Omron CX-Programmer project 新工程 (CX-Programmer 9.73)

# PLC 新PLC1: CPM2* 

## Global symbols (name address type ; comment)
0.00 BOOL  ; 外部急停
0.01 BOOL  ; 自动启动
0.02 BOOL  ; 手动封切
0.03 BOOL  ; 侧推反向磁环
0.04 BOOL  ; 侧推正向磁环
0.05 BOOL  ; 直推反向磁环
0.06 BOOL  ; 直推正向磁环
0.07 BOOL  ; 上膜接近开关
0.08 BOOL  ; 下膜接近开关
0.09 BOOL  ; 封口反向磁环
0.10 BOOL  ; 封口正向磁环
0.11 BOOL  ; 压料反向磁环
10.00 BOOL  ; 侧推电磁阀
10.01 BOOL  ; 直推电磁阀
10.02 BOOL  ; 封口电磁阀
10.03 BOOL  ; 切膜电磁阀
10.04 BOOL  ; 压料电磁阀
10.05 BOOL  ; 上膜电机
10.06 BOOL  ; 下膜电机
10.07 BOOL  ; 送料电机
11.00 BOOL  ; 后送料输出
11.01 BOOL  ; 浮动护栏气缸
11.02 BOOL  ; 一号气缸
11.03 BOOL  ; 二号气缸
11.04 BOOL  ; 三号气缸
11.05 BOOL  ; 四号气缸
11.06 BOOL  ; 熔接输出
11.07 BOOL  ; 熔接瞬间
12.00 BOOL  ; 加热
12.01 BOOL  ; 热风
12.02 BOOL  ; 后输送
12.03 BOOL  ; 报警输出
12.04 BOOL  ; 左右挡板电磁阀
12.05 BOOL  ; 前压料反向电磁阀
13 CHANNEL  ; 套膜包装控制寄存
13.00 BOOL  ; 直推
13.01 BOOL  ; 直推退回
13.02 BOOL  ; 封口
13.03 BOOL  ; 切膜
13.04 BOOL  ; 封膜
13.05 BOOL  ; 气缸复位
13.06 BOOL  ; 后送料启动
14 CHANNEL  ; 自动进料控制寄存
14.00 BOOL  ; 分层/挡料
14.01 BOOL  ; 左右挡板伸出
14.02 BOOL  ; 进料检测
14.03 BOOL  ; 左右挡板回位
14.04 BOOL  ; 顶料上升
14.05 BOOL  ; 末层判断
14.06 BOOL  ; 下一包挡料
14.07 BOOL  ; 左右挡板伸出
14.07 BOOL  ; 顶料下降
14.08 BOOL  ; 侧推
14.09 BOOL  ; 直推
14.10 BOOL  ; 侧推退回
14.11 BOOL  ; 进料完成
16 CHANNEL  ; 气缸输出
17.00 BOOL  ; 一号挡料板
17.01 BOOL  ; 二号挡料板
17.02 BOOL  ; 三号挡料板
17.03 BOOL  ; 四号挡料板
17.04 BOOL  ; 无挡料板
17.08 BOOL  ; 检测第一位
17.09 BOOL  ; 检测第二位
17.10 BOOL  ; 检测第三位
17.11 BOOL  ; 检测第四位
17.12 BOOL  ; 检测第五位
19 CHANNEL  ; 手动封切控制寄存
1.00 BOOL  ; 切膜反向磁环
1.01 BOOL  ; 浮动反向磁环
1.02 BOOL  ; 浮动正向磁环
1.03 BOOL  ; 一号正向磁环
1.04 BOOL  ; 二号正向磁环
1.05 BOOL  ; 三号正向磁环
1.06 BOOL  ; 四号正向磁环
1.07 BOOL  ; 检料光电01
1.08 BOOL  ; 检料光电02
1.09 BOOL  ; 检料接近11
1.10 BOOL  ; 检料接近12
1.11 BOOL  ; 检料光电21
204 CHANNEL  ; 临时整数
20.00 BOOL  ; 文本数据输入
20.01 BOOL  ; 文本数据初始化
20.02 BOOL  ; 文本收缩自动启动
20.03 BOOL  ; 文本收缩自动停止
20.04 BOOL  ; 文本手动封切
20.06 BOOL  ; 文本前送料
20.07 BOOL  ; 文本后送料
20.08 BOOL  ; 文本手动单次进料
20.09 BOOL  ; 文本直推料
20.10 BOOL  ; 文本封口
20.11 BOOL  ; 文本切膜
20.12 BOOL  ; 文本压料
20.13 BOOL  ; 文本自动开始
20.14 BOOL  ; 文本自动停止
20.15 BOOL  ; 文本复位
21.00 BOOL  ; 文本浮动护栏
21.01 BOOL  ; 文本一号气缸
21.02 BOOL  ; 文本二号气缸
21.03 BOOL  ; 文本三号气缸
21.04 BOOL  ; 文本四号气缸
21.05 BOOL  ; 左右气缸反向
21.06 BOOL  ; 文本前压料抬起
21.08 BOOL  ; 文本侧推料
23.00 BOOL  ; 文本加热
23.01 BOOL  ; 文本启用第六条延
23.02 BOOL  ; 文本使用第六条延
23.04 BOOL  ; 自动运行状态
23.05 BOOL  ; 远程启动
23.06 BOOL  ; 远程控制切换
23.07 BOOL  ; 接受控制
23.08 BOOL  ; 强制清除当前数据
23.10 BOOL  ; 文本风机
23.11 BOOL  ; 文本热风
23.13 BOOL  ; 文本输送
23.15 BOOL  ; 文本数据清除
24.00 BOOL  ; 校验不正确
24.02 BOOL  ; 远程不能启动
24.04 BOOL  ; 应答状态_急停
2.00 BOOL  ; 检料光电22
2.01 BOOL  ; 检料接近3
2.02 BOOL  ; 检料光电41
2.03 BOOL  ; 检料光电42
2.04 BOOL  ; 检料接近5
2.05 BOOL  ; 左右挡板正向磁环
2.06 BOOL  ; 左右挡板反向磁环
2.07 BOOL  ; 挡料板反向磁环2
2.08 BOOL  ; 挡料板反向磁环1
2.09 BOOL  ; 第7条
2.10 BOOL  ; 检料接近51
2.11 BOOL  ; 检料接近31
3.01 BOOL  ; 热风机保护
3.08 BOOL  ; 输送故障
3.09 BOOL  ; 前送料故障
3.10 BOOL  ; 后送料故障
3.11 BOOL  ; 超温报警输入
4.00 BOOL  ; 侧推输出
4.01 BOOL  ; 二号气缸输出
4.02 BOOL  ; 封口输出
4.03 BOOL  ; 浮动护栏输出
4.04 BOOL  ; 后压料输出
4.05 BOOL  ; 前压料放下
4.06 BOOL  ; 三号气缸输出
4.08 BOOL  ; 手动状态
4.09 BOOL  ; 四号气缸输出
4.10 BOOL  ; 一号气缸输出
4.11 BOOL  ; 直推输出
4.14 BOOL  ; 自动进料可以启动
DM2044 CHANNEL  ; 压料延时
HR0.02 BOOL  ; 不允许远程控制
TIM002 BOOL  ; 后送料定时器
TIM006 BOOL  ; 顶料延时
TIM011 BOOL  ; 前压料安全延时
TIM020 BOOL  ; 封口延时
TIM021 BOOL  ; 切膜延时
TIM022 BOOL  ; 封膜延时
TIM023 BOOL  ; 压料延时
TIM050 BOOL  ; 气缸推出定时器
TIM100 BOOL  ; 进料检测延时

## Program 新程序1 (no task)
; 这是一个用于食品包装生产线的立式包装机控制系统，通过PLC控制实现饼干的自动包装和封口。 / 系统采用CPM2*型号PLC控制器，连接送料电机、上膜电机、下膜电机、侧推电磁阀、直推电磁阀、封口电磁阀、切膜电磁阀、压料电磁阀、检料光电、接近开关和磁环等物理设备。 / 操作员按下自动启动后，系统进入自动模式。 / 检料光电01和检料光电02必须同时检测到饼干到位，送料电机才会启动，将饼干送入包装位置。 / 当检料光电01和检料光电02检测到物料时，产生物料到位信号。 / 随后，侧推电磁阀推动饼干对齐。在侧推正向磁环确认到位后，直推电磁阀动作，将饼干推入膜袋。 / 上膜电机和下膜电机分别在上膜接近开关和下膜接近开关触发时运行，确保膜材准确送入。 / 上膜接近开关触发时，启动上膜电机；下膜接近开关未触发时，启动下膜电机。 / 接着，封口电磁阀和切膜电磁阀执行封口和切膜，封口延时控制封口时间，若超时则通过报警输出警示操作员。 / 封口延时结束后，若封口未完成，触发报警输出。 / 完成后，后送料输出将成品送出生产线。 / 若生产线出现异常，外部急停触发时，侧推电磁阀、直推电磁阀、封口电磁阀、切膜电磁阀、压料电磁阀、上膜电机、下膜电机和送料电机会立即停止，确保人员和设备安全。 / 外部急停触发时，产生急停状态。 / 压料电磁阀由手动状态控制。 / 系统支持远程操作，但远程启动只有在不允许远程控制为假时生效。 / 远程启动触发时，激活远程操作信号。

### Section 段1

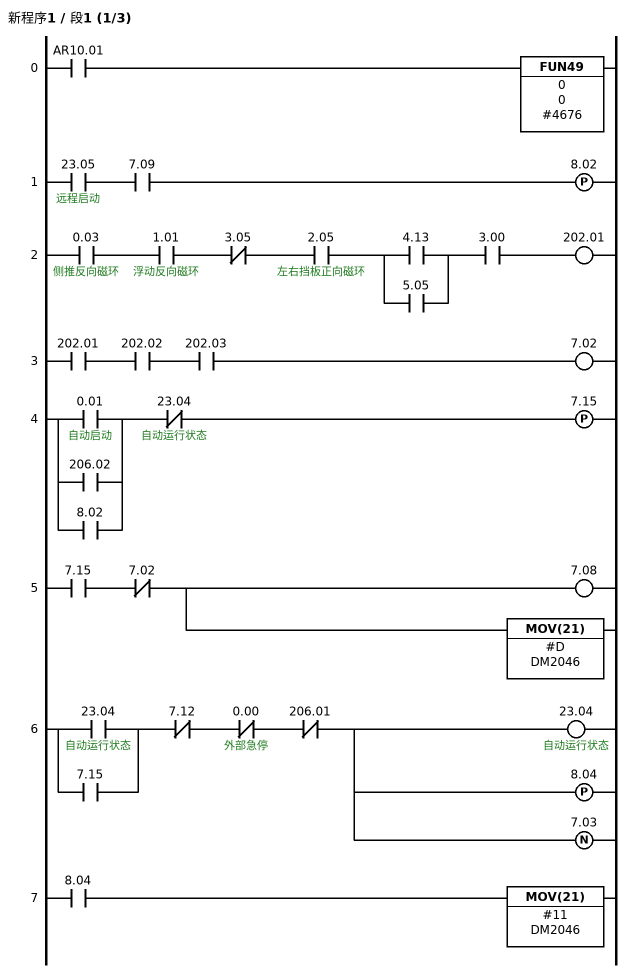
; rung 0
LD AR10.01
FUN49 0 0 #4676
; rung 1
LD 23.05  ; 远程启动
AND 7.09
DIFU(13) 8.02
; rung 2
LD 0.03  ; 侧推反向磁环
AND 1.01  ; 浮动反向磁环
ANDNOT 3.05
AND 2.05  ; 左右挡板正向磁环
LD 4.13
OR 5.05
ANDLD
AND 3.00
OUT 202.01
; rung 3
LD 202.01
AND 202.02
AND 202.03
OUT 7.02
; rung 4
LD 0.01  ; 自动启动
OR 206.02
OR 8.02
ANDNOT 23.04  ; 自动运行状态
DIFU(13) 7.15
; rung 5
LD 7.15
ANDNOT 7.02
OUT 7.08
MOV(21) #D DM2046
; rung 6
LD 23.04  ; 自动运行状态
OR 7.15
ANDNOT 7.12
ANDNOT 0.00  ; 外部急停
ANDNOT 206.01
OUT 23.04  ; 自动运行状态
DIFU(13) 8.04
DIFD(14) 7.03
; rung 7
LD 8.04
MOV(21) #11 DM2046

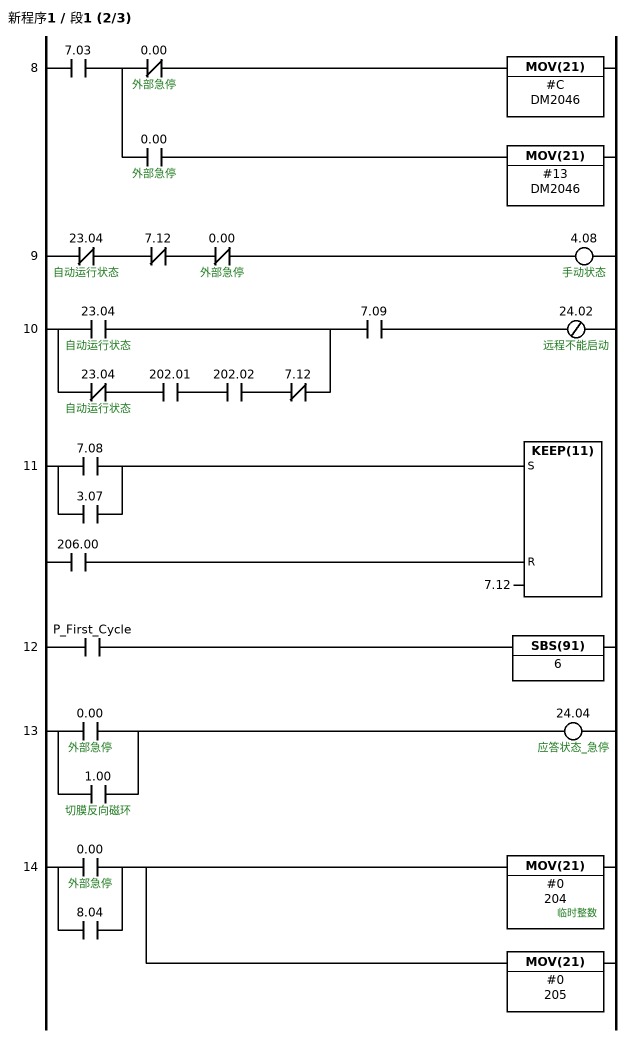
; rung 8
LD 7.03
OUT TR0
ANDNOT 0.00  ; 外部急停
MOV(21) #C DM2046
LD TR0
AND 0.00  ; 外部急停
MOV(21) #13 DM2046
; rung 9
LDNOT 23.04  ; 自动运行状态
ANDNOT 7.12
ANDNOT 0.00  ; 外部急停
OUT 4.08  ; 手动状态
; rung 10
LD 23.04  ; 自动运行状态
LDNOT 23.04  ; 自动运行状态
AND 202.01
AND 202.02
ANDNOT 7.12
ORLD
AND 7.09
OUTNOT 24.02  ; 远程不能启动
; rung 11
LD 7.08
OR 3.07
LD 206.00
KEEP(11) 7.12
; rung 12
LD P_First_Cycle
SBS(91) 6
; rung 13
LD 0.00  ; 外部急停
OR 1.00  ; 切膜反向磁环
OUT 24.04  ; 应答状态_急停
; rung 14
LD 0.00  ; 外部急停
OR 8.04
MOV(21) #0 204  ; 临时整数
MOV(21) #0 205

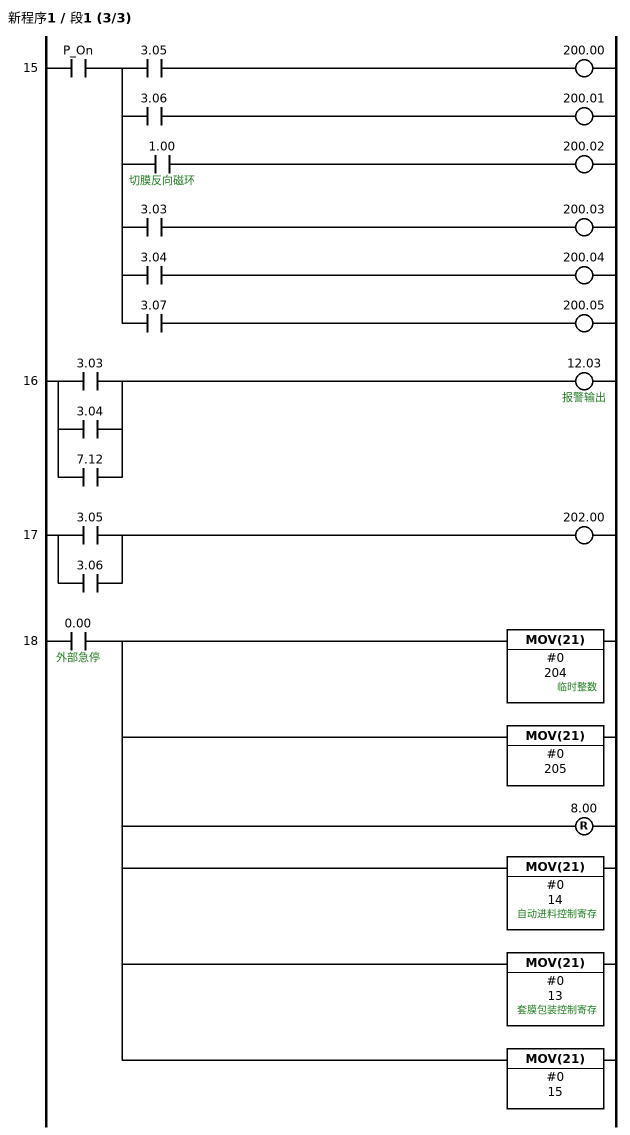
; rung 15
LD P_On
OUT TR0
AND 3.05
OUT 200.00
LD TR0
AND 3.06
OUT 200.01
LD TR0
AND 1.00  ; 切膜反向磁环
OUT 200.02
LD TR0
AND 3.03
OUT 200.03
LD TR0
AND 3.04
OUT 200.04
LD TR0
AND 3.07
OUT 200.05
; rung 16
LD 3.03
OR 3.04
OR 7.12
OUT 12.03  ; 报警输出
; rung 17
LD 3.05
OR 3.06
OUT 202.00
; rung 18
LD 0.00  ; 外部急停
MOV(21) #0 204  ; 临时整数
MOV(21) #0 205
RSET 8.00
MOV(21) #0 14  ; 自动进料控制寄存
MOV(21) #0 13  ; 套膜包装控制寄存
MOV(21) #0 15

### Section 段2

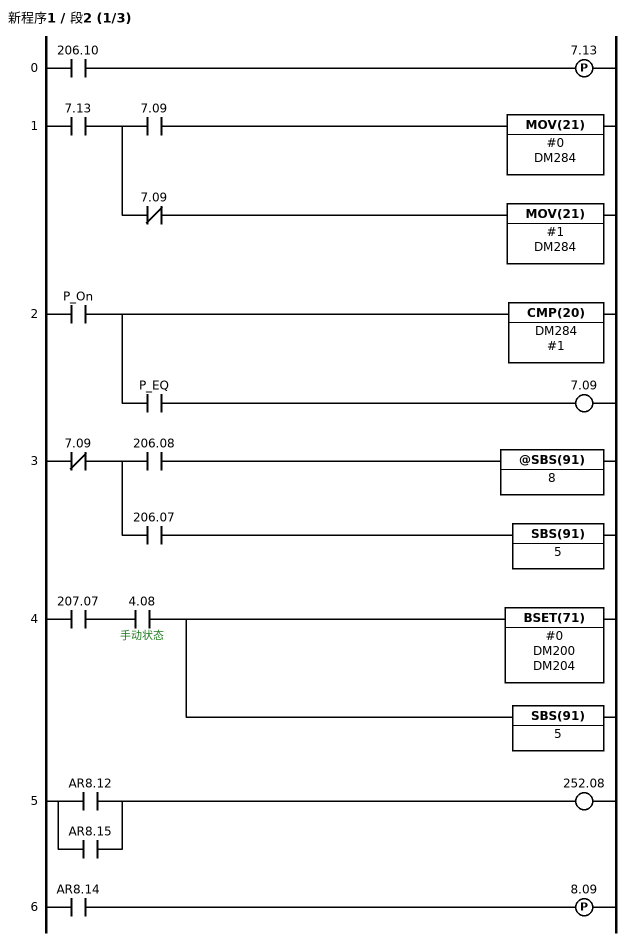
; rung 0
LD 206.10
DIFU(13) 7.13
; rung 1
LD 7.13
OUT TR0
AND 7.09
MOV(21) #0 DM284
LD TR0
ANDNOT 7.09
MOV(21) #1 DM284
; rung 2
LD P_On
CMP(20) DM284 #1
AND P_EQ
OUT 7.09
; rung 3
LDNOT 7.09
OUT TR0
AND 206.08
@SBS(91) 8
LD TR0
AND 206.07
SBS(91) 5
; rung 4
LD 207.07
AND 4.08  ; 手动状态
BSET(71) #0 DM200 DM204
SBS(91) 5
; rung 5
LD AR8.12
OR AR8.15
OUT 252.08
; rung 6
LD AR8.14
DIFU(13) 8.09

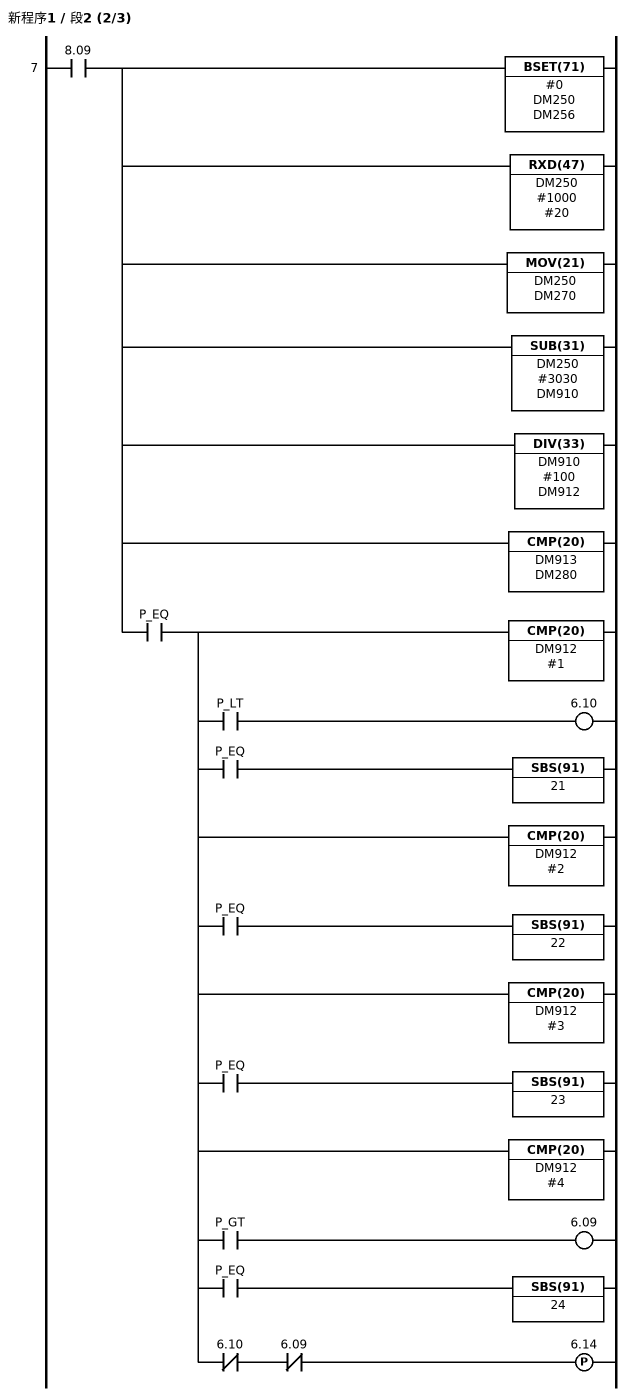
; rung 7
LD 8.09
BSET(71) #0 DM250 DM256
RXD(47) DM250 #1000 #20
MOV(21) DM250 DM270
SUB(31) DM250 #3030 DM910
DIV(33) DM910 #100 DM912
CMP(20) DM913 DM280
AND P_EQ
OUT TR0
CMP(20) DM912 #1
AND P_LT
OUT 6.10
LD TR0
AND P_EQ
SBS(91) 21
LD TR0
CMP(20) DM912 #2
AND P_EQ
SBS(91) 22
LD TR0
CMP(20) DM912 #3
AND P_EQ
SBS(91) 23
LD TR0
CMP(20) DM912 #4
AND P_GT
OUT 6.09
LD TR0
AND P_EQ
SBS(91) 24
LD TR0
ANDNOT 6.10
ANDNOT 6.09
DIFU(13) 6.14

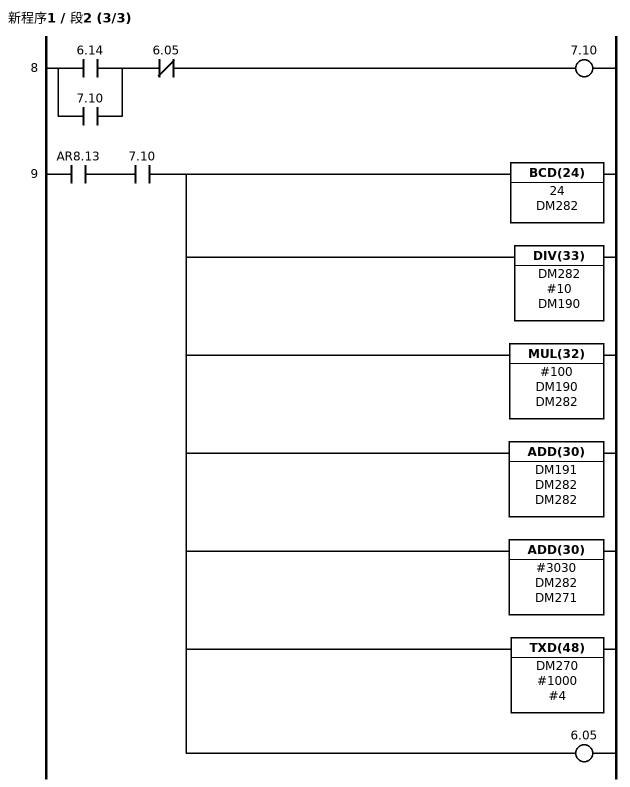
; rung 8
LD 6.14
OR 7.10
ANDNOT 6.05
OUT 7.10
; rung 9
LD AR8.13
AND 7.10
BCD(24) 24 DM282
DIV(33) DM282 #10 DM190
MUL(32) #100 DM190 DM282
ADD(30) DM191 DM282 DM282
ADD(30) #3030 DM282 DM271
TXD(48) DM270 #1000 #4
OUT 6.05

### Section 段3

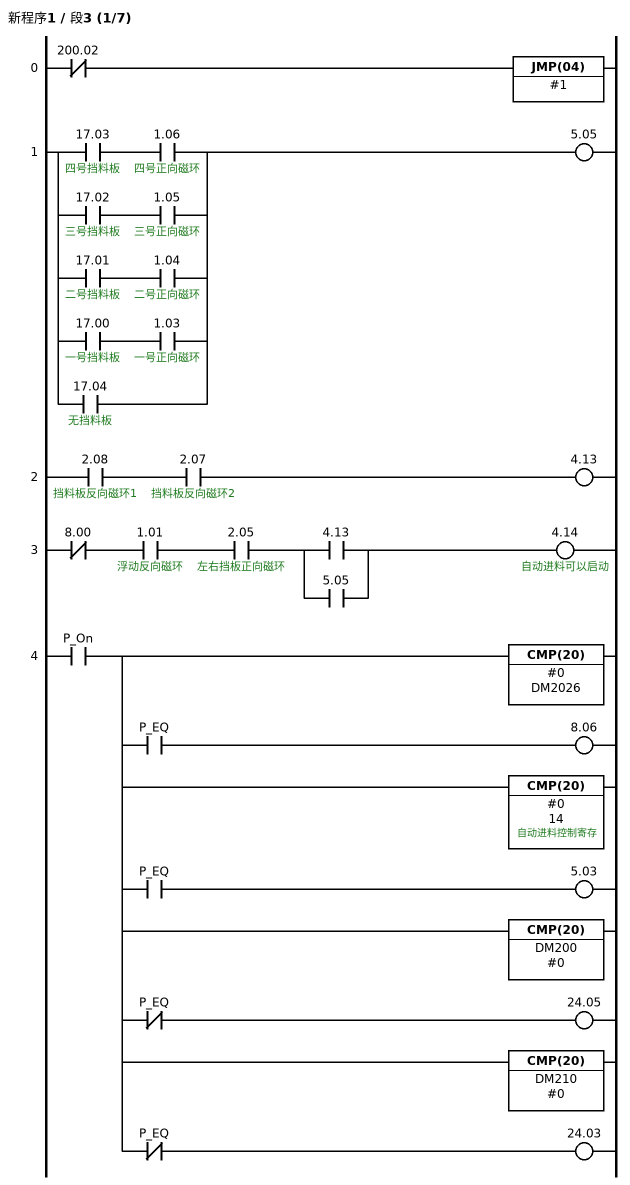
; rung 0
LDNOT 200.02
JMP(04) #1
; rung 1
LD 17.03  ; 四号挡料板
AND 1.06  ; 四号正向磁环
LD 17.02  ; 三号挡料板
AND 1.05  ; 三号正向磁环
ORLD
LD 17.01  ; 二号挡料板
AND 1.04  ; 二号正向磁环
ORLD
LD 17.00  ; 一号挡料板
AND 1.03  ; 一号正向磁环
ORLD
OR 17.04  ; 无挡料板
OUT 5.05
; rung 2
LD 2.08  ; 挡料板反向磁环1
AND 2.07  ; 挡料板反向磁环2
OUT 4.13
; rung 3
LDNOT 8.00
AND 1.01  ; 浮动反向磁环
AND 2.05  ; 左右挡板正向磁环
LD 4.13
OR 5.05
ANDLD
OUT 4.14  ; 自动进料可以启动
; rung 4
LD P_On
OUT TR0
CMP(20) #0 DM2026
AND P_EQ
OUT 8.06
LD TR0
CMP(20) #0 14  ; 自动进料控制寄存
AND P_EQ
OUT 5.03
LD TR0
CMP(20) DM200 #0
ANDNOT P_EQ
OUT 24.05
LD TR0
CMP(20) DM210 #0
ANDNOT P_EQ
OUT 24.03

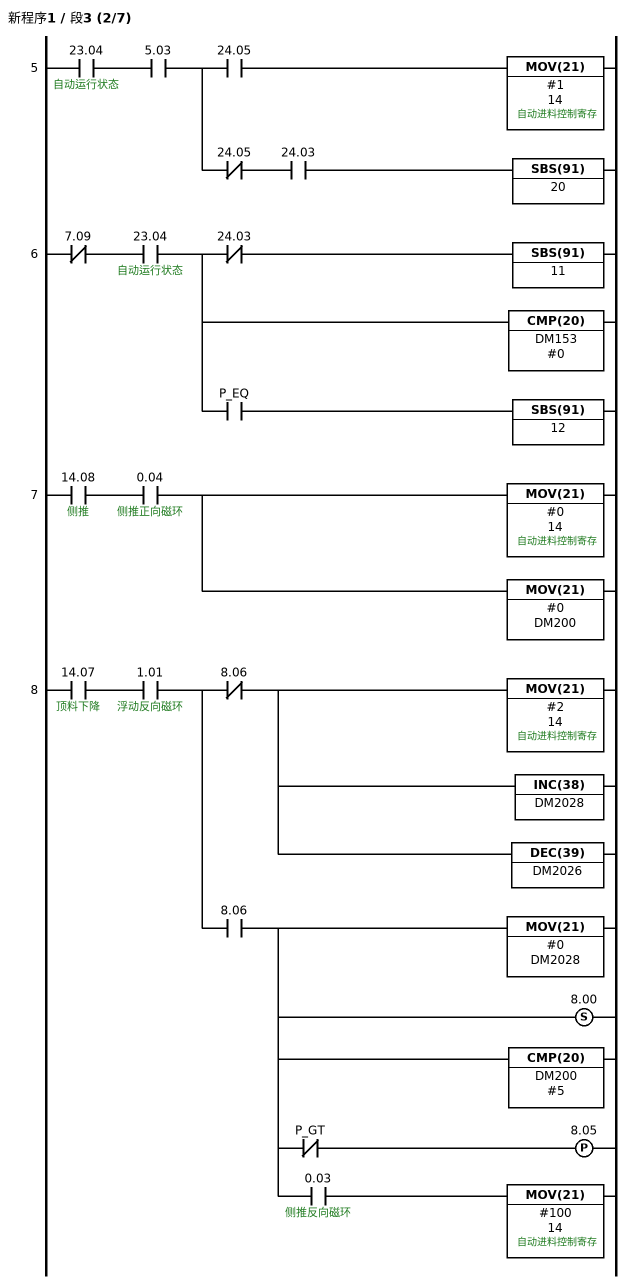
; rung 5
LD 23.04  ; 自动运行状态
AND 5.03
OUT TR0
AND 24.05
MOV(21) #1 14  ; 自动进料控制寄存
LD TR0
ANDNOT 24.05
AND 24.03
SBS(91) 20
; rung 6
LDNOT 7.09
AND 23.04  ; 自动运行状态
OUT TR0
ANDNOT 24.03
SBS(91) 11
LD TR0
CMP(20) DM153 #0
AND P_EQ
SBS(91) 12
; rung 7
LD 14.08  ; 侧推
AND 0.04  ; 侧推正向磁环
MOV(21) #0 14  ; 自动进料控制寄存
MOV(21) #0 DM200
; rung 8
LD 14.07  ; 顶料下降
AND 1.01  ; 浮动反向磁环
OUT TR0
ANDNOT 8.06
MOV(21) #2 14  ; 自动进料控制寄存
INC(38) DM2028
DEC(39) DM2026
LD TR0
AND 8.06
OUT TR0
MOV(21) #0 DM2028
SET 8.00
CMP(20) DM200 #5
ANDNOT P_GT
DIFU(13) 8.05
LD TR0
AND 0.03  ; 侧推反向磁环
MOV(21) #100 14  ; 自动进料控制寄存

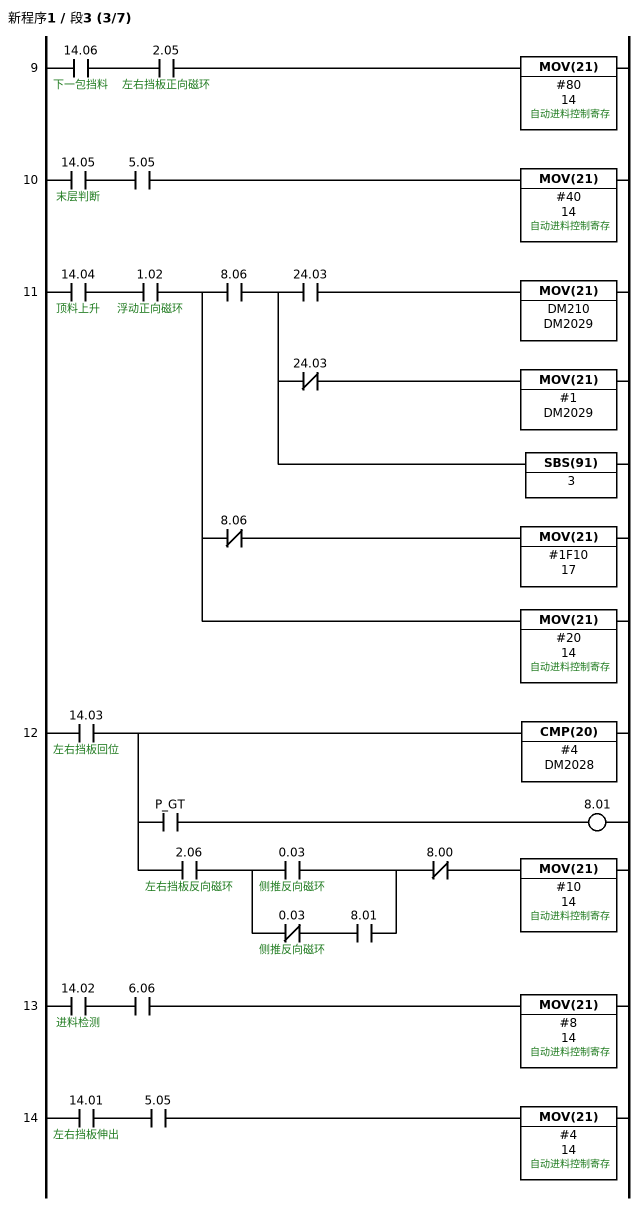
; rung 9
LD 14.06  ; 下一包挡料
AND 2.05  ; 左右挡板正向磁环
MOV(21) #80 14  ; 自动进料控制寄存
; rung 10
LD 14.05  ; 末层判断
AND 5.05
MOV(21) #40 14  ; 自动进料控制寄存
; rung 11
LD 14.04  ; 顶料上升
AND 1.02  ; 浮动正向磁环
OUT TR0
AND 8.06
OUT TR1
AND 24.03
MOV(21) DM210 DM2029
LD TR1
ANDNOT 24.03
MOV(21) #1 DM2029
LD TR1
SBS(91) 3
LD TR0
ANDNOT 8.06
MOV(21) #1F10 17
LD TR0
MOV(21) #20 14  ; 自动进料控制寄存
; rung 12
LD 14.03  ; 左右挡板回位
OUT TR0
CMP(20) #4 DM2028
AND P_GT
OUT 8.01
LD TR0
AND 2.06  ; 左右挡板反向磁环
LD 0.03  ; 侧推反向磁环
LDNOT 0.03  ; 侧推反向磁环
AND 8.01
ORLD
ANDLD
ANDNOT 8.00
MOV(21) #10 14  ; 自动进料控制寄存
; rung 13
LD 14.02  ; 进料检测
AND 6.06
MOV(21) #8 14  ; 自动进料控制寄存
; rung 14
LD 14.01  ; 左右挡板伸出
AND 5.05
MOV(21) #4 14  ; 自动进料控制寄存

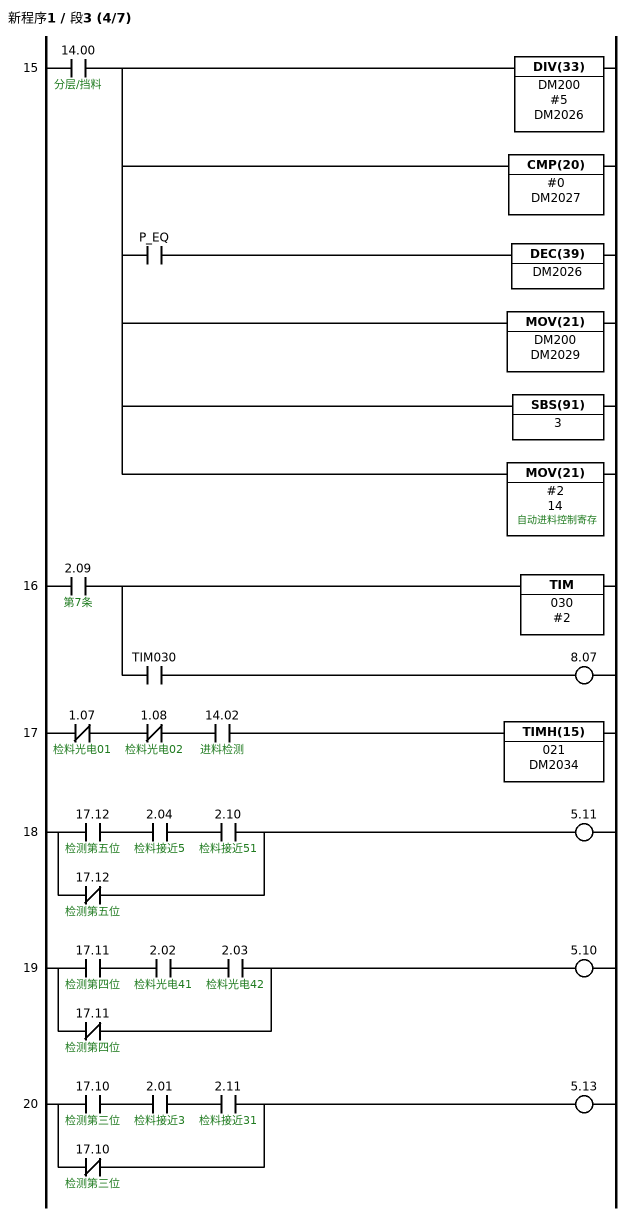
; rung 15
LD 14.00  ; 分层/挡料
OUT TR0
DIV(33) DM200 #5 DM2026
CMP(20) #0 DM2027
AND P_EQ
DEC(39) DM2026
LD TR0
MOV(21) DM200 DM2029
SBS(91) 3
MOV(21) #2 14  ; 自动进料控制寄存
; rung 16
LD 2.09  ; 第7条
TIM 030 #2
AND TIM030
OUT 8.07
; rung 17
LDNOT 1.07  ; 检料光电01
ANDNOT 1.08  ; 检料光电02
AND 14.02  ; 进料检测
TIMH(15) 021 DM2034
; rung 18
LD 17.12  ; 检测第五位
AND 2.04  ; 检料接近5
AND 2.10  ; 检料接近51
ORNOT 17.12  ; 检测第五位
OUT 5.11
; rung 19
LD 17.11  ; 检测第四位
AND 2.02  ; 检料光电41
AND 2.03  ; 检料光电42
ORNOT 17.11  ; 检测第四位
OUT 5.10
; rung 20
LD 17.10  ; 检测第三位
AND 2.01  ; 检料接近3
AND 2.11  ; 检料接近31
ORNOT 17.10  ; 检测第三位
OUT 5.13

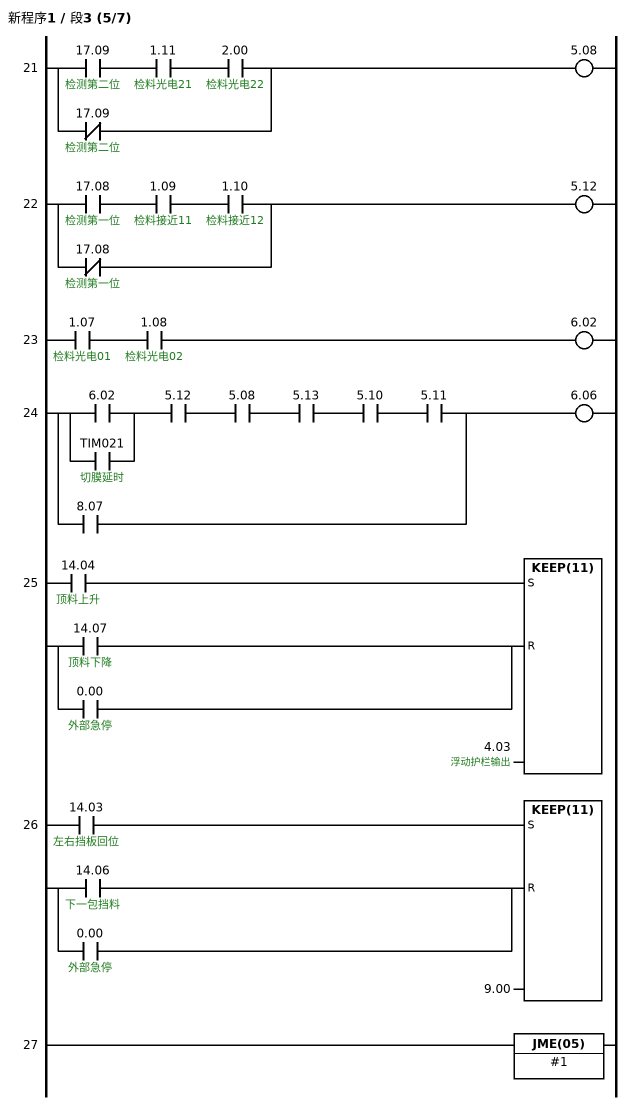
; rung 21
LD 17.09  ; 检测第二位
AND 1.11  ; 检料光电21
AND 2.00  ; 检料光电22
ORNOT 17.09  ; 检测第二位
OUT 5.08
; rung 22
LD 17.08  ; 检测第一位
AND 1.09  ; 检料接近11
AND 1.10  ; 检料接近12
ORNOT 17.08  ; 检测第一位
OUT 5.12
; rung 23
LD 1.07  ; 检料光电01
AND 1.08  ; 检料光电02
OUT 6.02
; rung 24
LD 6.02
OR TIM021  ; 切膜延时
AND 5.12
AND 5.08
AND 5.13
AND 5.10
AND 5.11
OR 8.07
OUT 6.06
; rung 25
LD 14.04  ; 顶料上升
LD 14.07  ; 顶料下降
OR 0.00  ; 外部急停
KEEP(11) 4.03  ; 浮动护栏输出
; rung 26
LD 14.03  ; 左右挡板回位
LD 14.06  ; 下一包挡料
OR 0.00  ; 外部急停
KEEP(11) 9.00
; rung 27
JME(05) #1

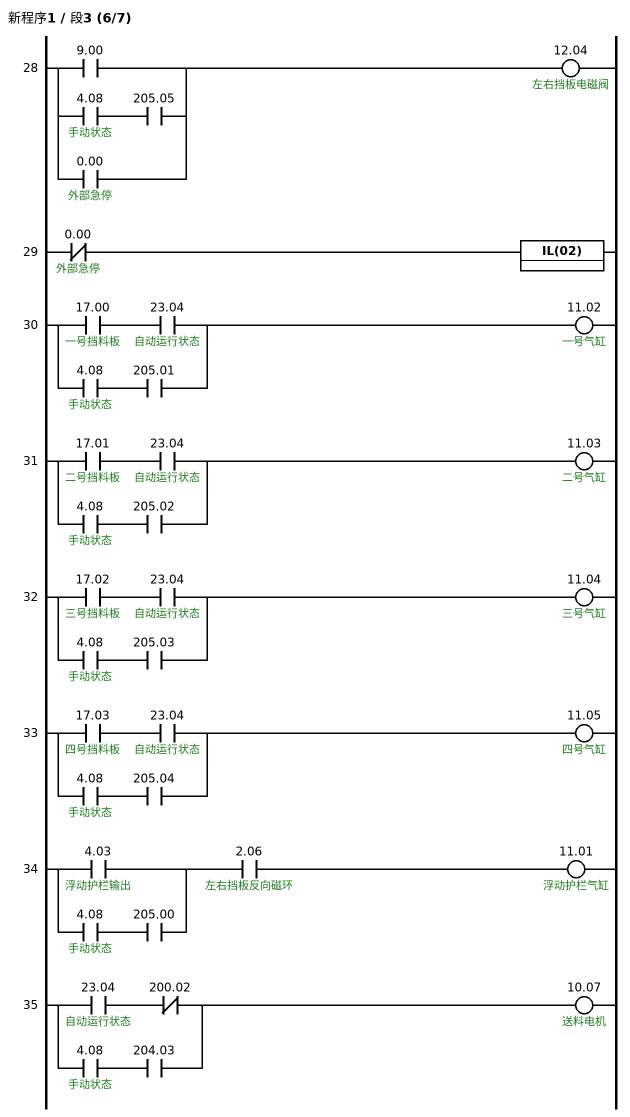
; rung 28
LD 9.00
LD 4.08  ; 手动状态
AND 205.05
ORLD
OR 0.00  ; 外部急停
OUT 12.04  ; 左右挡板电磁阀
; rung 29
LDNOT 0.00  ; 外部急停
IL(02)
; rung 30
LD 17.00  ; 一号挡料板
AND 23.04  ; 自动运行状态
LD 4.08  ; 手动状态
AND 205.01
ORLD
OUT 11.02  ; 一号气缸
; rung 31
LD 17.01  ; 二号挡料板
AND 23.04  ; 自动运行状态
LD 4.08  ; 手动状态
AND 205.02
ORLD
OUT 11.03  ; 二号气缸
; rung 32
LD 17.02  ; 三号挡料板
AND 23.04  ; 自动运行状态
LD 4.08  ; 手动状态
AND 205.03
ORLD
OUT 11.04  ; 三号气缸
; rung 33
LD 17.03  ; 四号挡料板
AND 23.04  ; 自动运行状态
LD 4.08  ; 手动状态
AND 205.04
ORLD
OUT 11.05  ; 四号气缸
; rung 34
LD 4.03  ; 浮动护栏输出
LD 4.08  ; 手动状态
AND 205.00
ORLD
AND 2.06  ; 左右挡板反向磁环
OUT 11.01  ; 浮动护栏气缸
; rung 35
LD 23.04  ; 自动运行状态
ANDNOT 200.02
LD 4.08  ; 手动状态
AND 204.03
ORLD
OUT 10.07  ; 送料电机

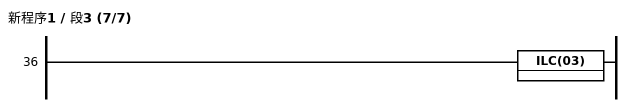
; rung 36
ILC(03)

### Section 段4

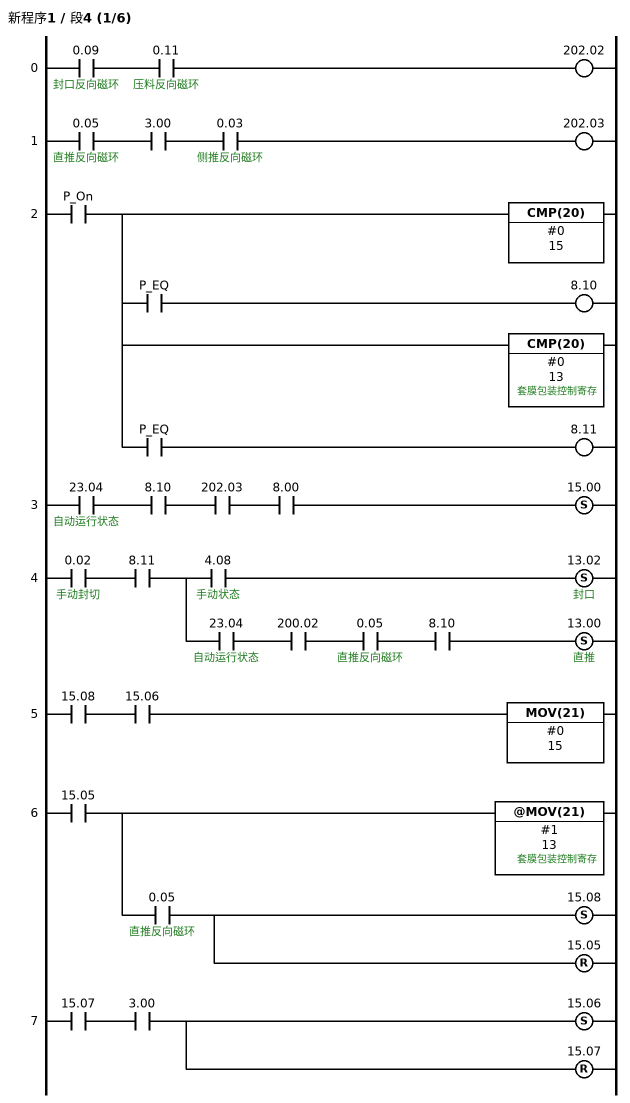
; rung 0
LD 0.09  ; 封口反向磁环
AND 0.11  ; 压料反向磁环
OUT 202.02
; rung 1
LD 0.05  ; 直推反向磁环
AND 3.00
AND 0.03  ; 侧推反向磁环
OUT 202.03
; rung 2
LD P_On
OUT TR0
CMP(20) #0 15
AND P_EQ
OUT 8.10
LD TR0
CMP(20) #0 13  ; 套膜包装控制寄存
AND P_EQ
OUT 8.11
; rung 3
LD 23.04  ; 自动运行状态
AND 8.10
AND 202.03
AND 8.00
SET 15.00
; rung 4
LD 0.02  ; 手动封切
AND 8.11
OUT TR0
AND 4.08  ; 手动状态
SET 13.02  ; 封口
LD TR0
AND 23.04  ; 自动运行状态
AND 200.02
AND 0.05  ; 直推反向磁环
AND 8.10
SET 13.00  ; 直推
; rung 5
LD 15.08
AND 15.06
MOV(21) #0 15
; rung 6
LD 15.05
@MOV(21) #1 13  ; 套膜包装控制寄存
AND 0.05  ; 直推反向磁环
SET 15.08
RSET 15.05
; rung 7
LD 15.07
AND 3.00
SET 15.06
RSET 15.07

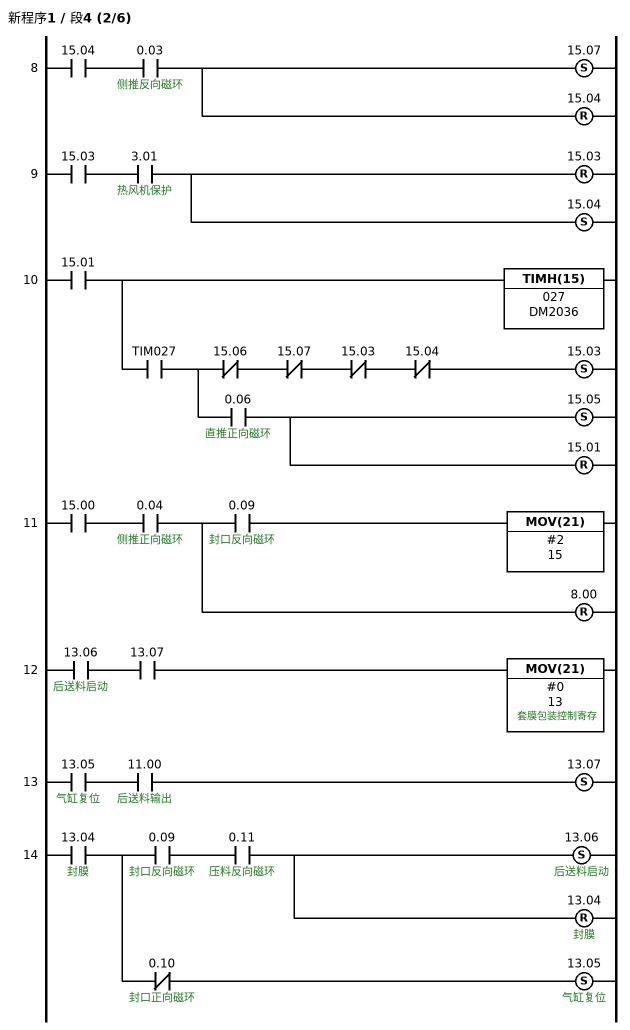
; rung 8
LD 15.04
AND 0.03  ; 侧推反向磁环
SET 15.07
RSET 15.04
; rung 9
LD 15.03
AND 3.01  ; 热风机保护
RSET 15.03
SET 15.04
; rung 10
LD 15.01
TIMH(15) 027 DM2036
AND TIM027
OUT TR0
ANDNOT 15.06
ANDNOT 15.07
ANDNOT 15.03
ANDNOT 15.04
SET 15.03
LD TR0
AND 0.06  ; 直推正向磁环
SET 15.05
RSET 15.01
; rung 11
LD 15.00
AND 0.04  ; 侧推正向磁环
OUT TR0
AND 0.09  ; 封口反向磁环
MOV(21) #2 15
LD TR0
RSET 8.00
; rung 12
LD 13.06  ; 后送料启动
AND 13.07
MOV(21) #0 13  ; 套膜包装控制寄存
; rung 13
LD 13.05  ; 气缸复位
AND 11.00  ; 后送料输出
SET 13.07
; rung 14
LD 13.04  ; 封膜
OUT TR0
AND 0.09  ; 封口反向磁环
AND 0.11  ; 压料反向磁环
SET 13.06  ; 后送料启动
RSET 13.04  ; 封膜
LD TR0
ANDNOT 0.10  ; 封口正向磁环
SET 13.05  ; 气缸复位

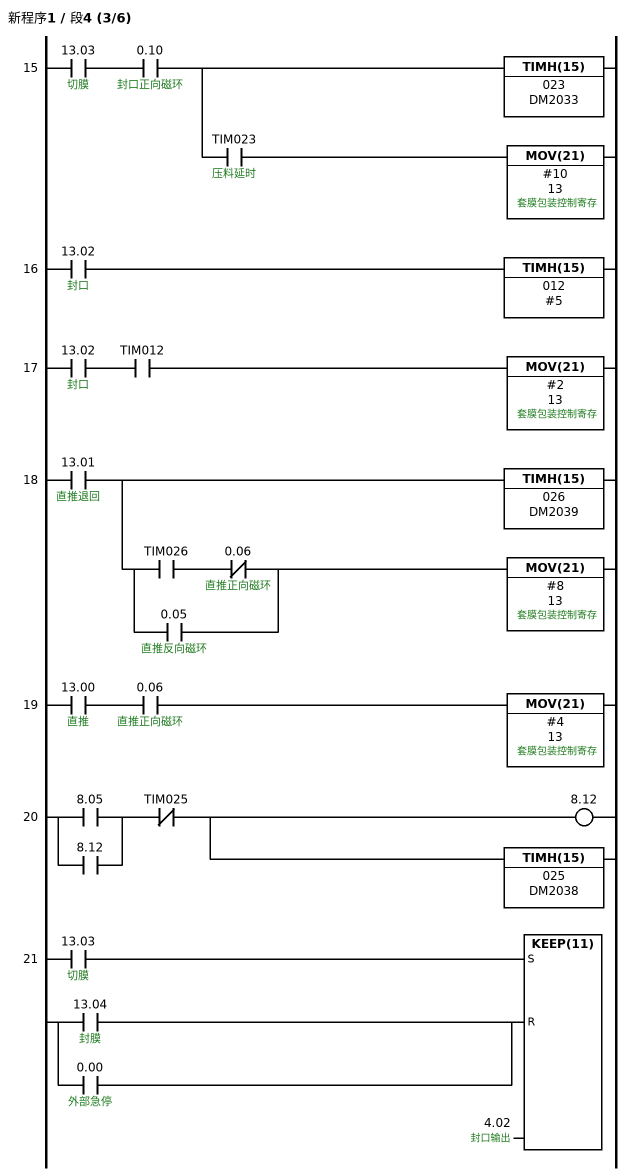
; rung 15
LD 13.03  ; 切膜
AND 0.10  ; 封口正向磁环
TIMH(15) 023 DM2033
AND TIM023  ; 压料延时
MOV(21) #10 13  ; 套膜包装控制寄存
; rung 16
LD 13.02  ; 封口
TIMH(15) 012 #5
; rung 17
LD 13.02  ; 封口
AND TIM012
MOV(21) #2 13  ; 套膜包装控制寄存
; rung 18
LD 13.01  ; 直推退回
TIMH(15) 026 DM2039
LD TIM026
ANDNOT 0.06  ; 直推正向磁环
OR 0.05  ; 直推反向磁环
ANDLD
MOV(21) #8 13  ; 套膜包装控制寄存
; rung 19
LD 13.00  ; 直推
AND 0.06  ; 直推正向磁环
MOV(21) #4 13  ; 套膜包装控制寄存
; rung 20
LD 8.05
OR 8.12
ANDNOT TIM025
OUT 8.12
TIMH(15) 025 DM2038
; rung 21
LD 13.03  ; 切膜
LD 13.04  ; 封膜
OR 0.00  ; 外部急停
KEEP(11) 4.02  ; 封口输出

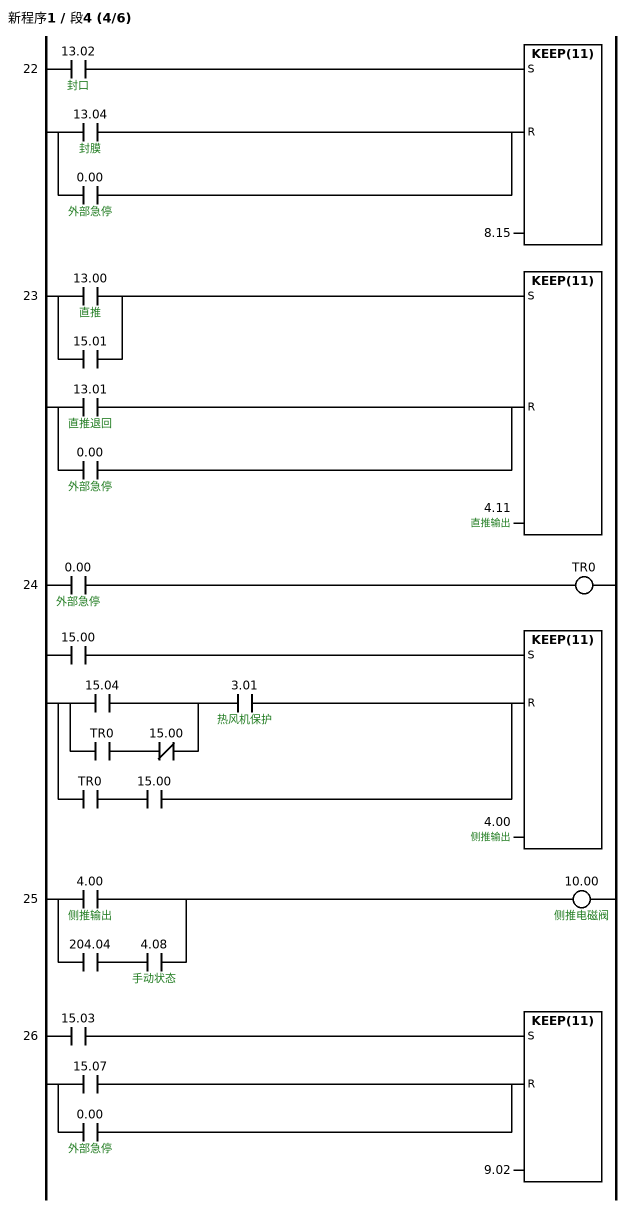
; rung 22
LD 13.02  ; 封口
LD 13.04  ; 封膜
OR 0.00  ; 外部急停
KEEP(11) 8.15
; rung 23
LD 13.00  ; 直推
OR 15.01
LD 13.01  ; 直推退回
OR 0.00  ; 外部急停
KEEP(11) 4.11  ; 直推输出
; rung 24
LD 15.00
LD 15.04
LD 0.00  ; 外部急停
OUT TR0
ANDNOT 15.00
ORLD
AND 3.01  ; 热风机保护
LD TR0
AND 15.00
ORLD
KEEP(11) 4.00  ; 侧推输出
; rung 25
LD 4.00  ; 侧推输出
LD 204.04
AND 4.08  ; 手动状态
ORLD
OUT 10.00  ; 侧推电磁阀
; rung 26
LD 15.03
LD 15.07
OR 0.00  ; 外部急停
KEEP(11) 9.02

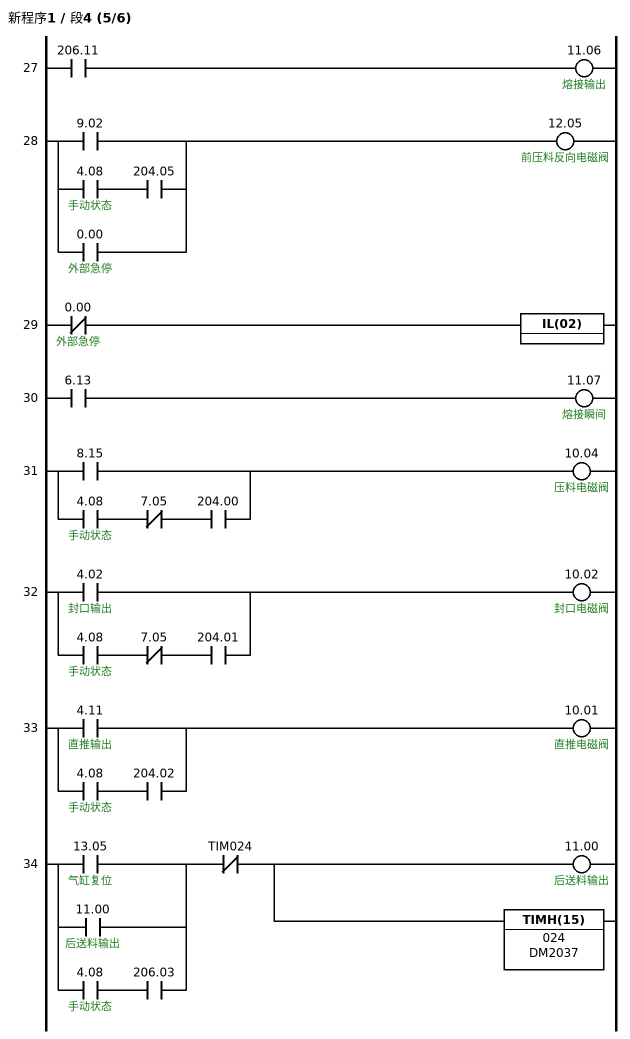
; rung 27
LD 206.11
OUT 11.06  ; 熔接输出
; rung 28
LD 9.02
LD 4.08  ; 手动状态
AND 204.05
ORLD
OR 0.00  ; 外部急停
OUT 12.05  ; 前压料反向电磁阀
; rung 29
LDNOT 0.00  ; 外部急停
IL(02)
; rung 30
LD 6.13
OUT 11.07  ; 熔接瞬间
; rung 31
LD 8.15
LD 4.08  ; 手动状态
ANDNOT 7.05
AND 204.00
ORLD
OUT 10.04  ; 压料电磁阀
; rung 32
LD 4.02  ; 封口输出
LD 4.08  ; 手动状态
ANDNOT 7.05
AND 204.01
ORLD
OUT 10.02  ; 封口电磁阀
; rung 33
LD 4.11  ; 直推输出
LD 4.08  ; 手动状态
AND 204.02
ORLD
OUT 10.01  ; 直推电磁阀
; rung 34
LD 13.05  ; 气缸复位
OR 11.00  ; 后送料输出
LD 4.08  ; 手动状态
AND 206.03
ORLD
ANDNOT TIM024
OUT 11.00  ; 后送料输出
TIMH(15) 024 DM2037

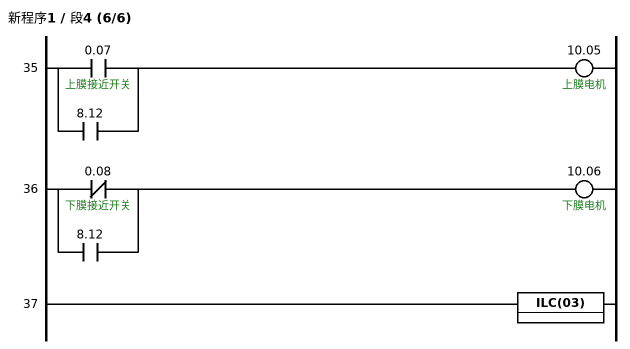
; rung 35
LD 0.07  ; 上膜接近开关
OR 8.12
OUT 10.05  ; 上膜电机
; rung 36
LDNOT 0.08  ; 下膜接近开关
OR 8.12
OUT 10.06  ; 下膜电机
; rung 37
ILC(03)

### Section 段5

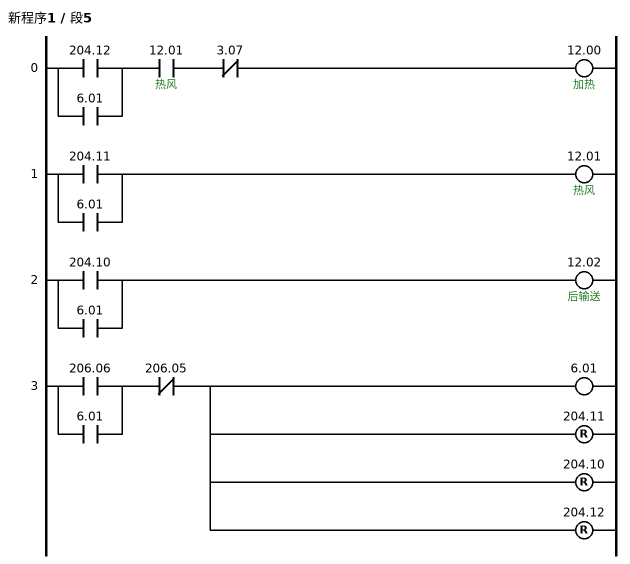
; rung 0
LD 204.12
OR 6.01
AND 12.01  ; 热风
ANDNOT 3.07
OUT 12.00  ; 加热
; rung 1
LD 204.11
OR 6.01
OUT 12.01  ; 热风
; rung 2
LD 204.10
OR 6.01
OUT 12.02  ; 后输送
; rung 3
LD 206.06
OR 6.01
ANDNOT 206.05
OUT 6.01
RSET 204.11
RSET 204.10
RSET 204.12

### Section 段6

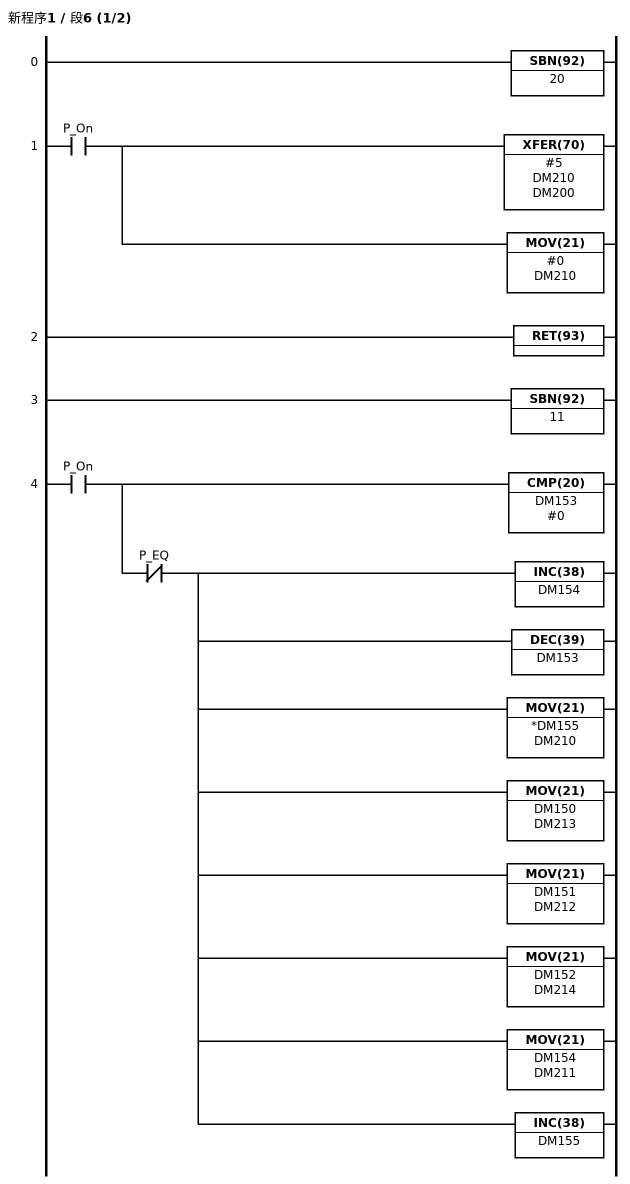
; rung 0
SBN(92) 20
; rung 1
LD P_On
XFER(70) #5 DM210 DM200
MOV(21) #0 DM210
; rung 2
RET(93)
; rung 3
SBN(92) 11
; rung 4
LD P_On
CMP(20) DM153 #0
ANDNOT P_EQ
INC(38) DM154
DEC(39) DM153
MOV(21) *DM155 DM210
MOV(21) DM150 DM213
MOV(21) DM151 DM212
MOV(21) DM152 DM214
MOV(21) DM154 DM211
INC(38) DM155

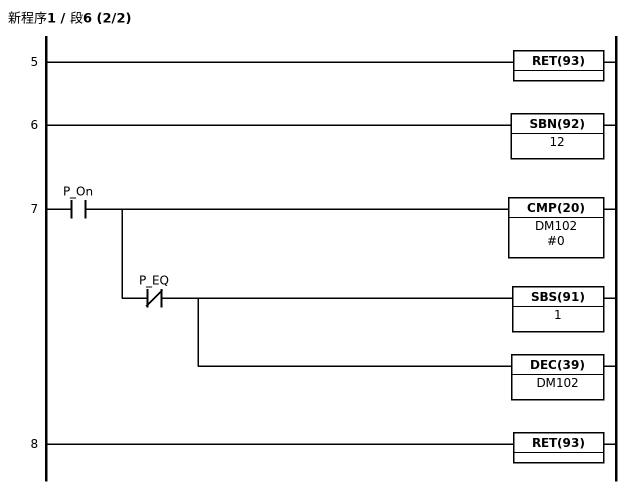
; rung 5
RET(93)
; rung 6
SBN(92) 12
; rung 7
LD P_On
CMP(20) DM102 #0
ANDNOT P_EQ
SBS(91) 1
DEC(39) DM102
; rung 8
RET(93)

### Section 段7

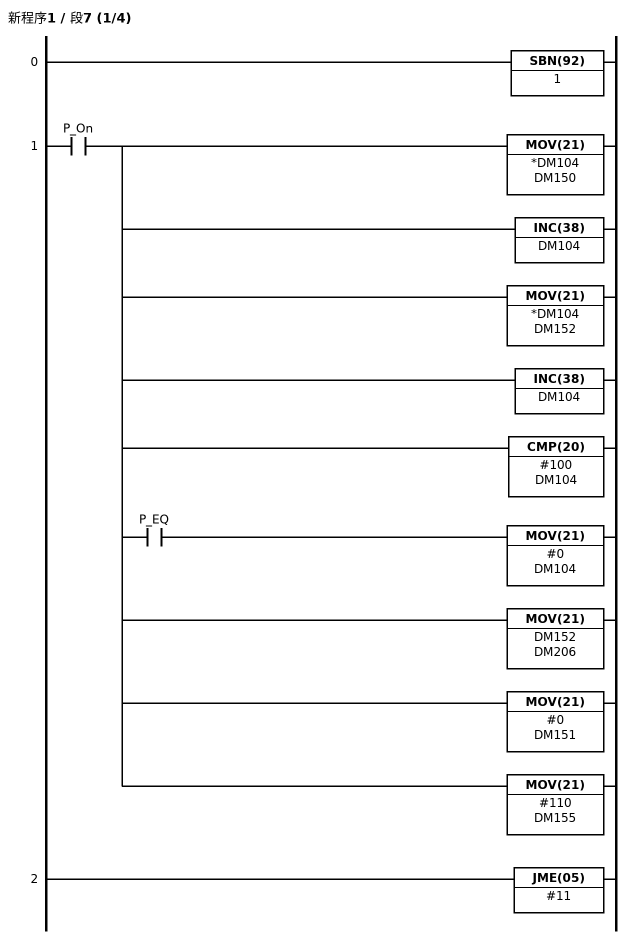
; rung 0
SBN(92) 1
; rung 1
LD P_On
OUT TR0
MOV(21) *DM104 DM150
INC(38) DM104
MOV(21) *DM104 DM152
INC(38) DM104
CMP(20) #100 DM104
AND P_EQ
MOV(21) #0 DM104
LD TR0
MOV(21) DM152 DM206
MOV(21) #0 DM151
MOV(21) #110 DM155
; rung 2
JME(05) #11

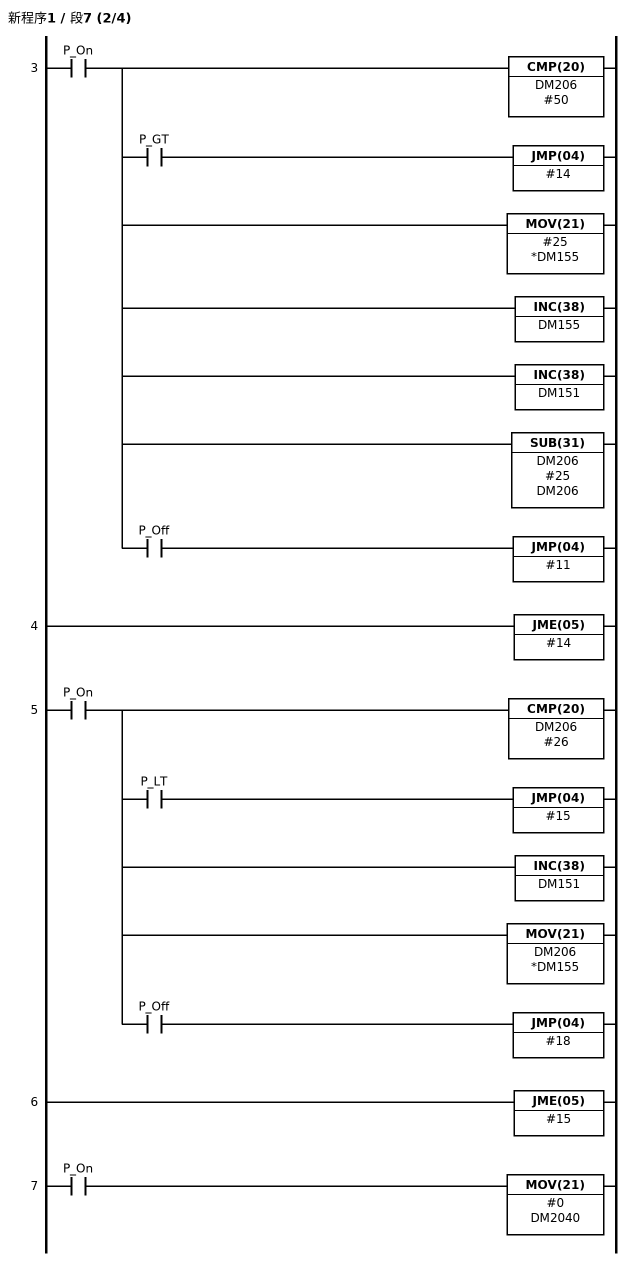
; rung 3
LD P_On
OUT TR0
CMP(20) DM206 #50
AND P_GT
JMP(04) #14
LD TR0
MOV(21) #25 *DM155
INC(38) DM155
INC(38) DM151
SUB(31) DM206 #25 DM206
AND P_Off
JMP(04) #11
; rung 4
JME(05) #14
; rung 5
LD P_On
OUT TR0
CMP(20) DM206 #26
AND P_LT
JMP(04) #15
LD TR0
INC(38) DM151
MOV(21) DM206 *DM155
AND P_Off
JMP(04) #18
; rung 6
JME(05) #15
; rung 7
LD P_On
MOV(21) #0 DM2040

